// TwinCAT 3 PLC project TcForgeReference
// Title: TcForgeReference
// Company: Home
// ProjectVersion: 2.0.0.0
// ProgramVersion: 3.1.4026.26
// libraries:
//   Tc2_Standard, 3.4.7.0 (Beckhoff Automation GmbH)
//   Tc2_System, 3.10.2.0 (Beckhoff Automation GmbH)
//   Tc3_Module, 3.4.7.0 (Beckhoff Automation GmbH)
//   [TcForge], 2.0.0.0 (Home)
// project tree:
//   TcForgeExample/Reference/ FB_ReferenceMachine.TcPOU, E_ReferenceCommand.TcDUT
//   Simulation/ FB_SimulationBridge.TcPOU
// (motion and I/O tree: see PLC project tcforge)
// real-time tasks:
//   TASK PlcTask: cycle T#10ms, priority 1, ADS port 350

// ---- TcForgeExample/Reference/E_ReferenceCommand.TcDUT
{attribute 'qualified_only'}
{attribute 'strict'}
TYPE E_ReferenceCommand : (None, Home, Start, Stop, Abort, Reset); END_TYPE

// ---- TcForgeExample/Reference/FB_ReferenceMachine.TcPOU
// Application composition. Call exactly once per scan from one owning task.
// No RPC entry points. command is sampled by this cyclic body on value changes.
FUNCTION_BLOCK FB_ReferenceMachine
VAR_INPUT
    // Explicit application policy for compatible engineering edits; gaps still cancel motion.
    recoverOnOnlineChange : BOOL := TRUE;
    command : E_ReferenceCommand;
    inAdvanced, inRetracted : BOOL;
    inputQuality : TcForge.E_IO_Quality := TcForge.E_IO_Quality.UNKNOWN;
    outputQuality : TcForge.E_IO_Quality := TcForge.E_IO_Quality.UNKNOWN;
    // Independent feedback from the application/plant, never synthesized from command bits.
    shutdownConfirmed : BOOL;
    shutdownQuality : TcForge.E_IO_Quality := TcForge.E_IO_Quality.UNKNOWN;
END_VAR
VAR_OUTPUT
    outAdvance, outRetract : BOOL;
    sequence : TcForge.ST_SM_Status;
    actuator : TcForge.ST_TwoPosActuator_Sts;
    faulted, qualityGood, outputsInhibited : BOOL;
    lastResponse : TcForge.E_RpcMethodResponse;
END_VAR
VAR
    continuity : TcForge.FB_ExecutionContinuity;
    taskIndex : DINT;
    recoveryRequired : BOOL;
    sm : TcForge.FB_StateMachine;
    clamp : TcForge.FB_TwoPosActuator;
    advanceOutput, retractOutput : TcForge.FB_DigitalOutput;
    homeStep, advanceStep, retractStep, stopCancelStep, stopRetractStep, abortStep : TcForge.FB_Step;
    previousCommand : E_ReferenceCommand;
    freshCommand, resetPending, confirmed, permitMotion : BOOL;
    response : TcForge.E_RpcMethodResponse;
END_VAR

// Execution interruption cancels intent before command admission or output evaluation.
taskIndex := Tc2_System.GETCURTASKINDEXEX();
IF taskIndex > 0 THEN
    continuity(taskIndex := taskIndex, cycleCounter := TwinCAT_SystemInfoVarList._TaskInfo[taskIndex].CycleCount,
        onlineChangeCounter := TwinCAT_SystemInfoVarList._AppInfo.OnlineChangeCnt,
        recoverOnOnlineChange := recoverOnOnlineChange);
ELSE continuity(taskIndex := taskIndex); END_IF;
IF continuity.interrupted THEN
    recoveryRequired := TRUE; sm.Abort(); clamp.Abort();
    advanceOutput.ForceSafe(); retractOutput.ForceSafe();
END_IF;
// 1. Sample quality and configure/map required conditions before any command.
qualityGood := inputQuality = TcForge.E_IO_Quality.GOOD AND outputQuality = TcForge.E_IO_Quality.GOOD;
confirmed := shutdownConfirmed AND shutdownQuality = TcForge.E_IO_Quality.GOOD;
sm.cfgHome.nRequired := 1; sm.cfgStart.nRequired := 1; sm.cfgAuto.nRequired := 1; sm.cfgRunning.nRequired := 1;
sm.MapHomeCondition(bitIndex := 0, bGood := qualityGood);
sm.MapStartCondition(bitIndex := 0, bGood := qualityGood);
sm.MapAutoCondition(bitIndex := 0, bGood := qualityGood);
sm.MapRunningIntlk(bitIndex := 0, bGood := qualityGood);
clamp.cfgAdvancePermissives.nRequired := 1; clamp.cfgRetractPermissives.nRequired := 1;
clamp.MapAdvanceCondition(bitIndex := 0, bGood := qualityGood);
clamp.MapRetractCondition(bitIndex := 0, bGood := qualityGood);
resetPending := FALSE;
freshCommand := command <> E_ReferenceCommand.None AND command <> previousCommand;
previousCommand := command;

IF freshCommand AND continuity.interrupted THEN
    lastResponse := TcForge.E_RpcMethodResponse.REJECTED_INTERLOCKED;
END_IF;
// 2. Commands are consumed once. A held or rejected command cannot become latent work.
IF freshCommand AND NOT continuity.interrupted THEN
    CASE command OF
    E_ReferenceCommand.Home:
        IF qualityGood AND NOT recoveryRequired THEN lastResponse := sm.Home(); ELSE lastResponse := TcForge.E_RpcMethodResponse.REJECTED_INTERLOCKED; END_IF;
    E_ReferenceCommand.Start:
        IF qualityGood AND NOT recoveryRequired THEN lastResponse := sm.Start(); ELSE lastResponse := TcForge.E_RpcMethodResponse.REJECTED_INTERLOCKED; END_IF;
    E_ReferenceCommand.Stop: lastResponse := sm.Stop();
    E_ReferenceCommand.Abort: lastResponse := sm.Abort();
    E_ReferenceCommand.Reset:
        IF sm.Status.State <> TcForge.E_SM_State.STOPPED THEN
            lastResponse := TcForge.E_RpcMethodResponse.REJECTED_WRONG_STATE;
        ELSIF NOT qualityGood OR NOT confirmed OR (inAdvanced AND inRetracted) THEN
            lastResponse := TcForge.E_RpcMethodResponse.REJECTED_INTERLOCKED;
        ELSE
            clamp.Reset(); advanceOutput.Reset(); retractOutput.Reset();
            sm.ResetRunningIntlk(); resetPending := TRUE;
        END_IF;
    ELSE lastResponse := TcForge.E_RpcMethodResponse.REJECTED_INVALID_PARAMETER;
    END_CASE;
END_IF;

// 3. State machine runs once, then every step once (including inactive steps).
sm(inpSubmoduleFaulted := clamp.IsFaulted() OR advanceOutput.IsFaulted() OR retractOutput.IsFaulted(), inpShutdownConfirmed := confirmed);
IF resetPending THEN
    lastResponse := sm.Reset();
    IF lastResponse = TcForge.E_RpcMethodResponse.ACCEPTED THEN recoveryRequired := FALSE; END_IF;
END_IF;

homeStep(sm := sm, nStep := 1000, nNextStep := 0, nRequired := 3, nTimeout := 6, sName := 'Retract clamp');
IF homeStep.Entry THEN
    response := clamp.Retract();
    IF response <> TcForge.E_RpcMethodResponse.ACCEPTED AND response <> TcForge.E_RpcMethodResponse.REJECTED_ALREADY_AT_TARGET THEN
        homeStep.RaiseFault(code := TcForge.E_SM_Fault.StepUserFault, reason := 'Clamp rejected motion command');
    END_IF;
END_IF;
IF homeStep.Execute THEN
    homeStep.MapPerm(nIndex := 0, sDescription := 'Position confirmed', bValue := inRetracted AND NOT inAdvanced);
    homeStep.MapPerm(nIndex := 1, sDescription := 'IO quality good', bValue := qualityGood);
END_IF;

advanceStep(sm := sm, nStep := 3000, nNextStep := 3002, nRequired := 3, nTimeout := 6, sName := 'Advance clamp');
IF advanceStep.Entry THEN
    response := clamp.Advance();
    IF response <> TcForge.E_RpcMethodResponse.ACCEPTED AND response <> TcForge.E_RpcMethodResponse.REJECTED_ALREADY_AT_TARGET THEN
        advanceStep.RaiseFault(code := TcForge.E_SM_Fault.StepUserFault, reason := 'Clamp rejected motion command');
    END_IF;
END_IF;
IF advanceStep.Execute THEN
    advanceStep.MapPerm(nIndex := 0, sDescription := 'Position confirmed', bValue := inAdvanced AND NOT inRetracted);
    advanceStep.MapPerm(nIndex := 1, sDescription := 'IO quality good', bValue := qualityGood);
END_IF;

retractStep(sm := sm, nStep := 3002, nNextStep := 0, nRequired := 3, nTimeout := 6, sName := 'Retract clamp');
IF retractStep.Entry THEN
    response := clamp.Retract();
    IF response <> TcForge.E_RpcMethodResponse.ACCEPTED AND response <> TcForge.E_RpcMethodResponse.REJECTED_ALREADY_AT_TARGET THEN
        retractStep.RaiseFault(code := TcForge.E_SM_Fault.StepUserFault, reason := 'Clamp rejected motion command');
    END_IF;
END_IF;
IF retractStep.Execute THEN
    retractStep.MapPerm(nIndex := 0, sDescription := 'Position confirmed', bValue := inRetracted AND NOT inAdvanced);
    retractStep.MapPerm(nIndex := 1, sDescription := 'IO quality good', bValue := qualityGood);
END_IF;

stopRetractStep(sm := sm, nStep := 2002, nNextStep := 0, nRequired := 3, nTimeout := 6, sName := 'Retract clamp');
IF stopRetractStep.Entry THEN
    response := clamp.Retract();
    IF response <> TcForge.E_RpcMethodResponse.ACCEPTED AND response <> TcForge.E_RpcMethodResponse.REJECTED_ALREADY_AT_TARGET THEN
        stopRetractStep.RaiseFault(code := TcForge.E_SM_Fault.StepUserFault, reason := 'Clamp rejected motion command');
    END_IF;
END_IF;
IF stopRetractStep.Execute THEN
    stopRetractStep.MapPerm(nIndex := 0, sDescription := 'Position confirmed', bValue := inRetracted AND NOT inAdvanced);
    stopRetractStep.MapPerm(nIndex := 1, sDescription := 'IO quality good', bValue := qualityGood);
END_IF;

stopCancelStep(sm := sm, nStep := 2000, nNextStep := 2002, nRequired := 0, nTimeout := 2, sName := 'Cancel motion before retract');
IF stopCancelStep.Entry THEN clamp.Abort(); END_IF;
abortStep(sm := sm, nStep := 5000, nNextStep := 0, nRequired := 1, nTimeout := 2, sName := 'Confirm shutdown');
IF abortStep.Entry THEN clamp.Abort(); END_IF;
IF abortStep.Execute THEN abortStep.MapPerm(nIndex := 0, sDescription := 'Independent shutdown feedback', bValue := confirmed); END_IF;

// 4. Monitor the actuator with this scan's feedback and permissives.
// Inhibition also cancels internal motion so stale intent cannot reappear later.
permitMotion := qualityGood AND NOT recoveryRequired AND NOT sm.IsFaulted() AND NOT sm.Status.ShutdownFailed AND
    (sm.Status.State = TcForge.E_SM_State.HOMING OR sm.Status.State = TcForge.E_SM_State.RUNNING OR sm.Status.State = TcForge.E_SM_State.STOPPING);
IF NOT permitMotion THEN clamp.Abort(); END_IF;
clamp(inAdvanced := inAdvanced, inRetracted := inRetracted);

// 5. Final output policy runs AFTER all fault detection and lifecycle commands.
permitMotion := permitMotion AND NOT clamp.IsFaulted() AND NOT advanceOutput.IsFaulted() AND NOT retractOutput.IsFaulted();
IF permitMotion THEN
    IF clamp.outAdvance THEN advanceOutput.SetOn(); ELSE advanceOutput.SetOff(); END_IF;
    IF clamp.outRetract THEN retractOutput.SetOn(); ELSE retractOutput.SetOff(); END_IF;
ELSE
    advanceOutput.ForceSafe(); retractOutput.ForceSafe();
END_IF;
advanceOutput(inpQuality := outputQuality); retractOutput(inpQuality := outputQuality);
outAdvance := advanceOutput.outSignal; outRetract := retractOutput.outSignal;
outputsInhibited := NOT permitMotion;
faulted := sm.IsFaulted() OR clamp.IsFaulted() OR advanceOutput.IsFaulted() OR retractOutput.IsFaulted();
sequence := sm.Status; actuator := clamp.sts;

END_FUNCTION_BLOCK

// ---- Simulation/FB_SimulationBridge.TcPOU
// Isolated simulation composition: no physical IO mapping and no persistent sessions.
FUNCTION_BLOCK FB_SimulationBridge
VAR_INPUT recoverOnOnlineChange : BOOL := TRUE; END_VAR
VAR_OUTPUT
    outAdvance, outRetract : BOOL;
END_VAR
VAR
    continuity : TcForge.FB_ExecutionContinuity;
    machine : FB_ReferenceMachine;
    mutex : BOOL;
    boot, cycle, session, submitted, applied, lastAck : ULINT;
    pending, hasFrame, freshPrevious, newClaim : BOOL;
    pendingAdvanced, pendingRetracted, pendingShutdown, pendingQuality : BOOL;
    advanced, retracted, shutdown, good : BOOL;
    pendingCommand : UINT;
    command : E_ReferenceCommand;
    quality : TcForge.E_IO_Quality;
    watchdog : TON;
    owner : DINT;
    ownershipConflict : BOOL;
END_VAR

// All exchange state and timer updates share the same bounded lock.
IF NOT Tc2_System.TestAndSet(mutex) THEN RETURN; END_IF;
IF owner = 0 THEN
    owner := Tc2_System.GETCURTASKINDEXEX();
    IF owner <= 0 THEN owner := 0; mutex := FALSE; RETURN; END_IF;
    boot := Tc2_System.F_GetSystemTime();
END_IF;
IF Tc2_System.GETCURTASKINDEXEX() <> owner THEN
    ownershipConflict := TRUE; session := 0; pending := FALSE; hasFrame := FALSE;
    outAdvance := FALSE; outRetract := FALSE; mutex := FALSE; RETURN;
END_IF;
// Gaps always invalidate sessions; compatible online edits follow explicit application policy.
continuity(taskIndex := owner, cycleCounter := TwinCAT_SystemInfoVarList._TaskInfo[owner].CycleCount,
    onlineChangeCounter := TwinCAT_SystemInfoVarList._AppInfo.OnlineChangeCnt,
    recoverOnOnlineChange := recoverOnOnlineChange);
IF continuity.interrupted THEN
    boot := Tc2_System.F_GetSystemTime();
    session := 0; pending := FALSE; hasFrame := FALSE; freshPrevious := FALSE; newClaim := FALSE;
    submitted := 0; applied := 0; lastAck := 0; pendingCommand := 0;
    watchdog(IN := FALSE, PT := T#250MS);
END_IF;
// Only the owning cyclic task advances the timer; RPCs never call the machine.
watchdog(IN := session <> 0 AND NOT freshPrevious, PT := T#250MS);
freshPrevious := FALSE;
IF newClaim THEN watchdog(IN := FALSE, PT := T#250MS); newClaim := FALSE; END_IF;
IF watchdog.Q OR ownershipConflict THEN
    session := 0; pending := FALSE; hasFrame := FALSE;
END_IF;
command := E_ReferenceCommand.None;
IF pending AND session <> 0 THEN
    advanced := pendingAdvanced; retracted := pendingRetracted;
    shutdown := pendingShutdown; good := pendingQuality;
    CASE pendingCommand OF
    1: command := E_ReferenceCommand.Home;
    2: command := E_ReferenceCommand.Start;
    3: command := E_ReferenceCommand.Stop;
    4: command := E_ReferenceCommand.Abort;
    5: command := E_ReferenceCommand.Reset;
    END_CASE;
    applied := submitted; pending := FALSE; hasFrame := TRUE; freshPrevious := TRUE;
END_IF;
IF hasFrame AND session <> 0 AND good AND NOT ownershipConflict THEN
    quality := TcForge.E_IO_Quality.GOOD;
ELSE quality := TcForge.E_IO_Quality.BAD;
END_IF;
// The canonical machine executes on every available PLC scan, never in RPC context.
machine(command := command, recoverOnOnlineChange := recoverOnOnlineChange,
    inAdvanced := advanced, inRetracted := retracted,
    inputQuality := quality, outputQuality := quality,
    shutdownConfirmed := shutdown, shutdownQuality := quality);
outAdvance := machine.outAdvance AND quality = TcForge.E_IO_Quality.GOOD;
outRetract := machine.outRetract AND quality = TcForge.E_IO_Quality.GOOD;
cycle := cycle + 1;
mutex := FALSE;

{attribute 'TcRpcEnable' := '1'}
METHOD PUBLIC Identity : STRING(80)
Identity := 'TcForge.DiscreteSimulation/1';
END_METHOD

{attribute 'TcRpcEnable' := '1'}
METHOD PUBLIC Claim : DINT
VAR_INPUT client : ULINT; expectedBoot : ULINT; END_VAR
Claim := 30;
IF client = 0 THEN RETURN; END_IF;
Claim := 22; IF NOT Tc2_System.TestAndSet(mutex) THEN RETURN; END_IF;
IF boot = 0 OR owner = 0 THEN Claim := 12;
ELSIF ownershipConflict THEN Claim := 13;
ELSIF expectedBoot <> boot THEN Claim := 34;
ELSIF session <> 0 THEN
    IF client = session THEN Claim := 0; ELSE Claim := 11; END_IF;
ELSE
    session := client; submitted := 0; applied := 0; lastAck := 0;
    pending := FALSE; hasFrame := FALSE; newClaim := TRUE; Claim := 0;
END_IF;
mutex := FALSE;
END_METHOD

{attribute 'TcRpcEnable' := '1'}
METHOD PUBLIC Exchange : DINT
VAR_INPUT
    client, expectedBoot, frame, outputFrame : ULINT;
    inAdvanced, inRetracted, shutdownConfirmed, qualityGood : BOOL;
    requestedCommand : UINT;
END_VAR
Exchange := 30;
IF client = 0 OR frame = 0 OR requestedCommand > 5 THEN RETURN; END_IF;
Exchange := 22; IF NOT Tc2_System.TestAndSet(mutex) THEN RETURN; END_IF;
IF expectedBoot <> boot THEN Exchange := 34;
ELSIF session = 0 OR watchdog.Q THEN Exchange := 12;
ELSIF client <> session THEN Exchange := 11;
ELSIF frame <= submitted THEN Exchange := 35;
ELSIF frame <> submitted + 1 OR outputFrame <= lastAck OR outputFrame > cycle THEN Exchange := 30;
ELSIF NOT pending THEN
    pendingAdvanced := inAdvanced; pendingRetracted := inRetracted;
    pendingShutdown := shutdownConfirmed; pendingQuality := qualityGood;
    pendingCommand := requestedCommand; submitted := frame; lastAck := outputFrame;
    pending := TRUE; Exchange := 1;
END_IF;
mutex := FALSE;
END_METHOD

{attribute 'TcRpcEnable' := '1'}
METHOD PUBLIC Release : DINT
VAR_INPUT client, expectedBoot : ULINT; END_VAR
Release := 22; IF NOT Tc2_System.TestAndSet(mutex) THEN RETURN; END_IF;
IF expectedBoot <> boot THEN Release := 34;
ELSIF session = 0 OR client <> session THEN Release := 11;
ELSE
    session := 0; hasFrame := FALSE; pending := FALSE;
    Release := 0;
END_IF;
mutex := FALSE;
END_METHOD

{attribute 'TcRpcEnable' := '1'}
METHOD PUBLIC Snapshot : STRING(255)
Snapshot := '22'; IF NOT Tc2_System.TestAndSet(mutex) THEN RETURN; END_IF;
Snapshot := '0';
Snapshot := CONCAT(Snapshot, CONCAT(',', ULINT_TO_STRING(boot)));
Snapshot := CONCAT(Snapshot, CONCAT(',', ULINT_TO_STRING(cycle)));
Snapshot := CONCAT(Snapshot, CONCAT(',', ULINT_TO_STRING(applied)));
Snapshot := CONCAT(Snapshot, CONCAT(',', DINT_TO_STRING(BOOL_TO_UINT(outAdvance))));
Snapshot := CONCAT(Snapshot, CONCAT(',', DINT_TO_STRING(BOOL_TO_UINT(outRetract))));
Snapshot := CONCAT(Snapshot, CONCAT(',', DINT_TO_STRING(machine.sequence.State)));
Snapshot := CONCAT(Snapshot, CONCAT(',', DINT_TO_STRING(BOOL_TO_UINT(machine.faulted))));
Snapshot := CONCAT(Snapshot, CONCAT(',', DINT_TO_STRING(BOOL_TO_UINT(machine.outputsInhibited))));
Snapshot := CONCAT(Snapshot, CONCAT(',', DINT_TO_STRING(machine.lastResponse)));
Snapshot := CONCAT(Snapshot, CONCAT(',', ULINT_TO_STRING(session)));
Snapshot := CONCAT(Snapshot, CONCAT(',', DINT_TO_STRING(owner)));
Snapshot := CONCAT(Snapshot, CONCAT(',', DINT_TO_STRING(BOOL_TO_UINT(quality = TcForge.E_IO_Quality.GOOD AND NOT watchdog.Q))));
mutex := FALSE;
END_METHOD

END_FUNCTION_BLOCK
